PROGRAM MAIN
VAR
	test : STRING := 'hello'; //this is a test variable to place in the textbox on the HMI
	//SAFE
	HoldButton : BOOL := FALSE;
	HoldSwitchLight : BOOL;
	SwitchButton : BOOL := FALSE;
	SwitchButtonLight : BOOL;
	
	StopButton : BOOL;

	Options : DropdownBox;
END_VAR

HoldSwitchLight:=HoldButton;
SwitchButtonLight:=SwitchButton;

IF StopButton THEN
	HoldButton:=FALSE;
	SwitchButton:=FALSE;
END_IF

END_PROGRAM

(* stored: Version 1.1.0.1, ProductVersion 3.1.4024.12
   POU MAIN: Id {95fa86a7-2031-4ef9-9bc3-09dd08f854df}, SpecialFunc None *)
